PROGRAM main
  VAR_INPUT
    IceRequest : BOOL;
    MixType1 : BOOL;
    MixType2 : BOOL;
    MixType3 : BOOL;
    Liqueur1 : BOOL;
    Liqueur2 : BOOL;
    WaterRequest : BOOL;
  END_VAR
  VAR_OUTPUT
    DispenseIce : BOOL;
    DispenseMix1 : BOOL;
    DispenseMix2 : BOOL;
    DispenseMix3 : BOOL;
    DispenseLiqueur1 : BOOL;
    DispenseLiqueur2 : BOOL;
    DispenseWater : BOOL;
    CocktailReady : BOOL;
  END_VAR

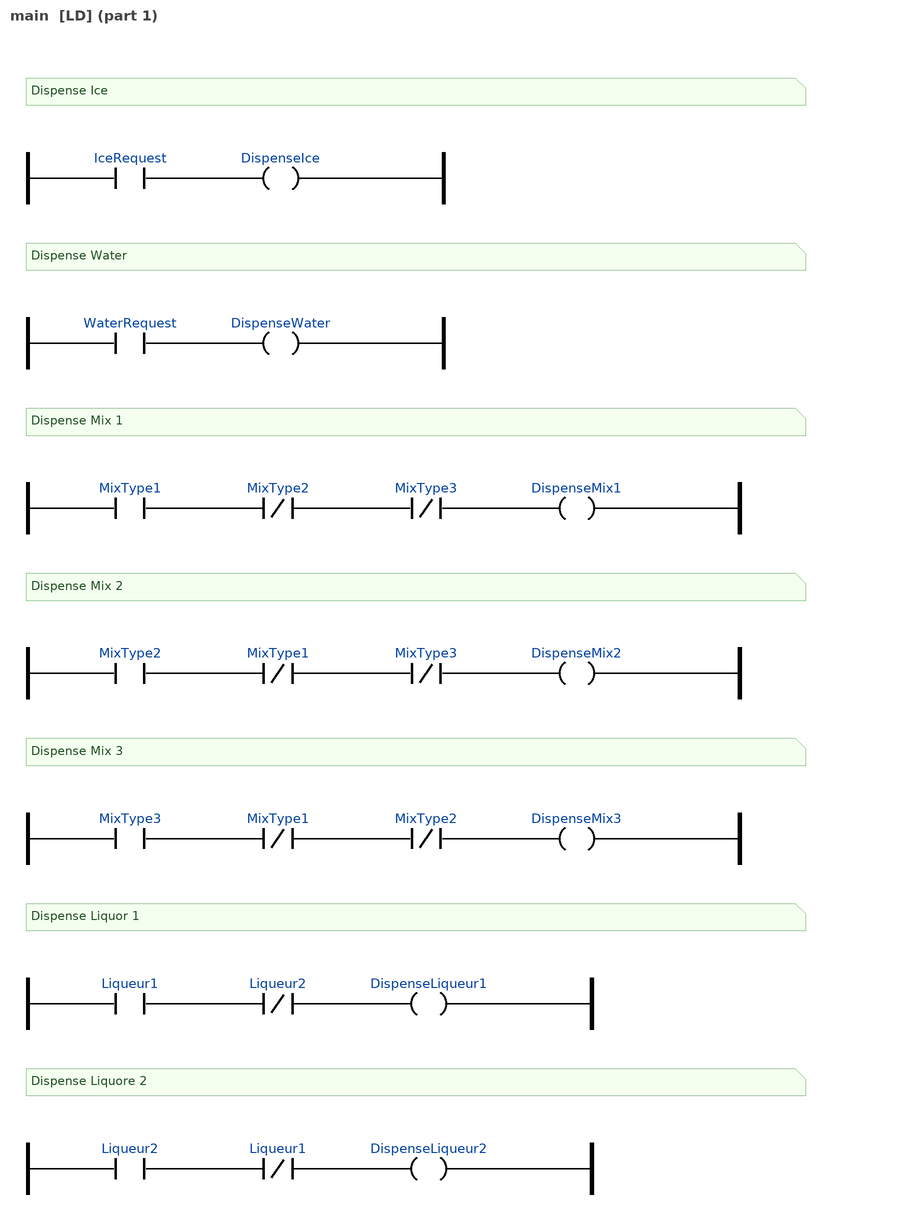
(* LD diagram, written out as Structured Text *)
(* Dispense Ice *)
DispenseIce := IceRequest;
(* Dispense Water *)
DispenseWater := WaterRequest;
(* Dispense Mix 1 *)
DispenseMix1 := MixType1 AND NOT MixType2 AND NOT MixType3;
(* Dispense Mix 2 *)
DispenseMix2 := MixType2 AND NOT MixType1 AND NOT MixType3;
(* Dispense Mix 3 *)
DispenseMix3 := MixType3 AND NOT MixType1 AND NOT MixType2;
(* Dispense Liquor 1 *)
DispenseLiqueur1 := Liqueur1 AND NOT Liqueur2;
(* Dispense Liquore 2 *)
DispenseLiqueur2 := Liqueur2 AND NOT Liqueur1;
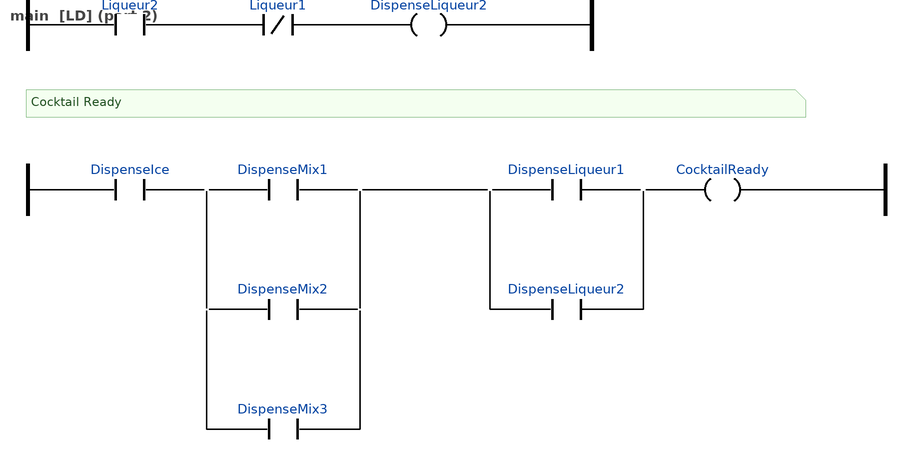
(* Cocktail Ready *)
CocktailReady := DispenseIce AND (DispenseMix1 OR DispenseMix2 OR DispenseMix3) AND (DispenseLiqueur1 OR DispenseLiqueur2);
END_PROGRAM
